FUNCTION F_CreateObjectName : STRING
VAR_INPUT
	strObjecktPath: STRING;
END_VAR
VAR
	strTemp: STRING;
	i: INT;
END_VAR


strTemp:=strObjecktPath;

FOR i:=1 TO 10 BY 1 DO
	IF FIND(strTemp,'.')>0 THEN
		strTemp:=DELETE(strTemp,FIND(strTemp,'.')+1,0);
	ELSE
		EXIT;
	END_IF
END_FOR

IF left(strTemp,2)='fb' THEN
	strTemp:=DELETE(strTemp,3,0);
END_IF

F_CreateObjectName:=strTemp;

END_FUNCTION

(* stored: Version 1.1.0.1, ProductVersion 3.1.4024.12
   POU F_CreateObjectName: Id {e2199058-f767-4f4e-801b-87e5fa8f2ba6}, SpecialFunc None *)
